Staubli VAL3: setConveyor.pgx

program setConveyor(num x_nConvNum (dimensions=1), frame& x_fFrame (dimensions=1))
begin
  switch x_nConvNum
    case 0
      call cnv0:setConveyor(x_fFrame)
    break
    case 1
      call cnv1:setConveyor(x_fFrame)
    break
  endSwitch
end
